(* PLC project CoDeSys External Library Template, WAGO e!COCKPIT e!COCKPIT, author 3S - Smart Software Solutions GmbH *)
(* stored: creationDateTime 2019-10-29T12:22:40.9320685, version 3.5.5.30, modificationDateTime 2019-10-24T14:40:07.960949, organization 3S - Smart Software Solutions GmbH *)
(* Library project template with all possible element types, docu and a sample project structure *)

FUNCTION fnKonwersja4x128na512 : BOOL
  VAR_INPUT
    sKomunikatCzesc1 : STRING(128);
    sKomunikatCzesc2 : STRING(128);
    sKomunikatCzesc3 : STRING(128);
    sKomunikatCzesc4 : STRING(128);
  END_VAR
  VAR_IN_OUT
    sKomunikat512 : alSTRINGKomunikat;
  END_VAR

            sKomunikat512 := CONCAT(sKomunikatCzesc1 , sKomunikatCzesc2);
sKomunikat512 := CONCAT(sKomunikat512 , sKomunikatCzesc3);
sKomunikat512 := CONCAT(sKomunikat512 , sKomunikatCzesc4);
          
END_FUNCTION
